// SIMATIC STEP 7 (V5.x) project parking2
// CPU: CPU 314C-2 DP
// station: Hardware
// station: SIMATIC 300(1)
// station: P_ADR_BUS
// program: S7 Program(2)

SYMBOL_TABLE
"res"	I 0.0	BOOL	// КжЮЭ ИСдЗге
"active"	I 0.5	BOOL	// ЭЪЗб УЗТ ИСдЗге
"enter"	I 0.6	BOOL	// ФУКн жСжПн
"exit"	I 0.7	BOOL	// ФУКн ОСжМн
"red light"	Q 0.0	BOOL
"yellow light"	Q 0.1	BOOL
"green light"	Q 0.2	BOOL
"light floor 1"	Q 1.0	BOOL
"light floor 2"	Q 1.1	BOOL
"light floor 3"	Q 1.2	BOOL
"parking is full"	Q 1.3	BOOL
"fan 1"	Q 1.4	BOOL	// floor 1
"fan 2"	Q 1.5	BOOL	// floor 1
"fan 3"	Q 1.6	BOOL	// floor 1
"fan 4"	Q 1.7	BOOL	// floor 1
"fan 5"	Q 2.0	BOOL	// floor 2
"fan 6"	Q 2.1	BOOL	// floor 2
"fan 7"	Q 2.2	BOOL	// floor 2
"fan 8"	Q 2.3	BOOL	// floor 2
"fan 9"	Q 2.4	BOOL	// floor 3
"fan 10"	Q 2.5	BOOL	// floor 3
"fan 11"	Q 2.6	BOOL	// floor 3
"fan 12"	Q 2.7	BOOL	// floor 3
END_SYMBOL_TABLE

ORGANIZATION_BLOCK OB 1
TITLE = "Main Program Sweep (Cycle)"
VERSION : 0.1
VAR_TEMP
  OB1_EV_CLASS : BYTE ;	//Bits 0-3 = 1 (Coming event), Bits 4-7 = 1 (Event class 1)
  OB1_SCAN_1 : BYTE ;	//1 (Cold restart scan 1 of OB 1), 3 (Scan 2-n of OB 1)
  OB1_PRIORITY : BYTE ;	//Priority of OB Execution
  OB1_OB_NUMBR : BYTE ;	//1 (Organization block 1, OB1)
  OB1_RESERVED_1 : BYTE ;	//Reserved for system
  OB1_RESERVED_2 : BYTE ;	//Reserved for system
  OB1_PREV_CYCLE : INT ;	//Cycle time of previous OB1 scan (milliseconds)
  OB1_MIN_CYCLE : INT ;	//Minimum cycle time of OB1 (milliseconds)
  OB1_MAX_CYCLE : INT ;	//Maximum cycle time of OB1 (milliseconds)
  OB1_DATE_TIME : DATE_AND_TIME ;	//Date and time OB1 started
END_VAR
BEGIN
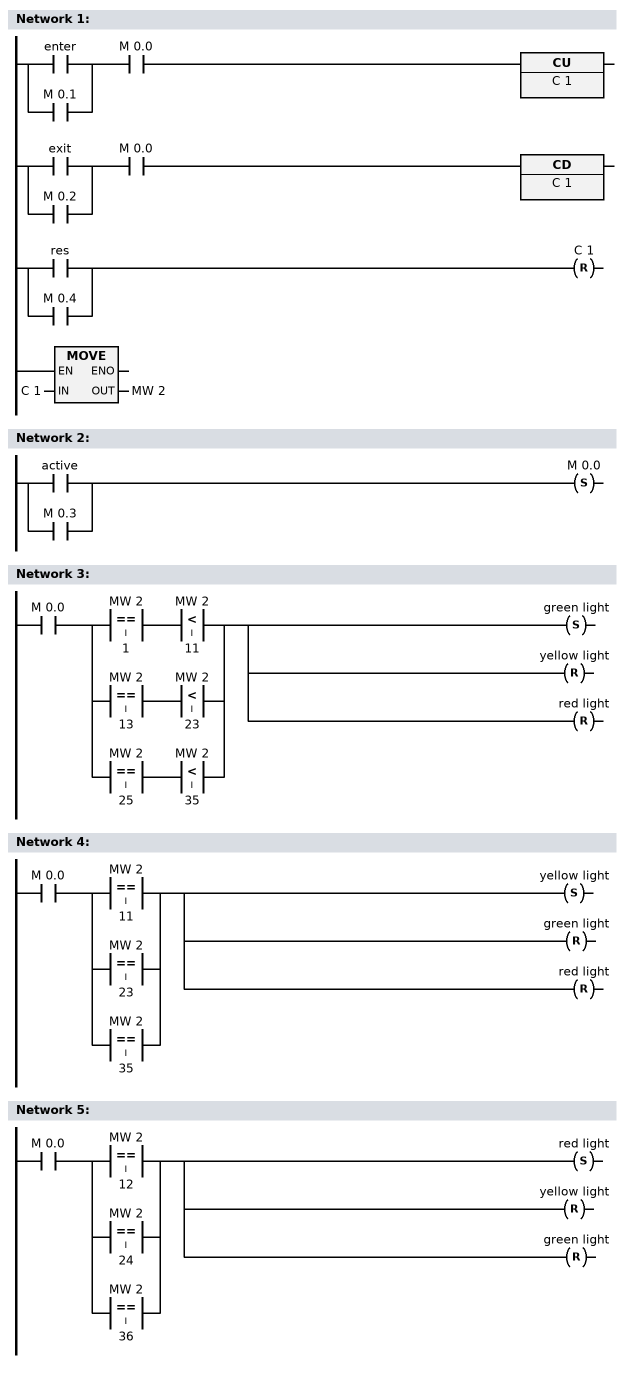
NETWORK
TITLE =
      A(;
      O     "enter";
      O     M 0.1;
      );
      A     M 0.0;
      CU    C 1;
      A(;
      O     "exit";
      O     M 0.2;
      );
      A     M 0.0;
      CD    C 1;
      NOP   0;
      NOP   0;
      A(;
      O     "res";
      O     M 0.4;
      );
      R     C 1;
      L     C 1;
      T     MW 2;
      NOP   0;
      NOP   0;
NETWORK
TITLE =
      O     "active";
      O     M 0.3;
      S     M 0.0;
NETWORK
TITLE =
      A     M 0.0;
      A(;
      A(;
      L     MW 2;
      L     1;
      ==I;
      );
      A(;
      L     MW 2;
      L     11;
      <I;
      );
      O;
      A(;
      L     MW 2;
      L     13;
      ==I;
      );
      A(;
      L     MW 2;
      L     23;
      <I;
      );
      O;
      A(;
      L     MW 2;
      L     25;
      ==I;
      );
      A(;
      L     MW 2;
      L     35;
      <I;
      );
      );
      S     "green light";
      R     "yellow light";
      R     "red light";
NETWORK
TITLE =
      A     M 0.0;
      A(;
      O(;
      L     MW 2;
      L     11;
      ==I;
      );
      O(;
      L     MW 2;
      L     23;
      ==I;
      );
      O(;
      L     MW 2;
      L     35;
      ==I;
      );
      );
      S     "yellow light";
      R     "green light";
      R     "red light";
NETWORK
TITLE =
      A     M 0.0;
      A(;
      O(;
      L     MW 2;
      L     12;
      ==I;
      );
      O(;
      L     MW 2;
      L     24;
      ==I;
      );
      O(;
      L     MW 2;
      L     36;
      ==I;
      );
      );
      S     "red light";
      R     "yellow light";
      R     "green light";
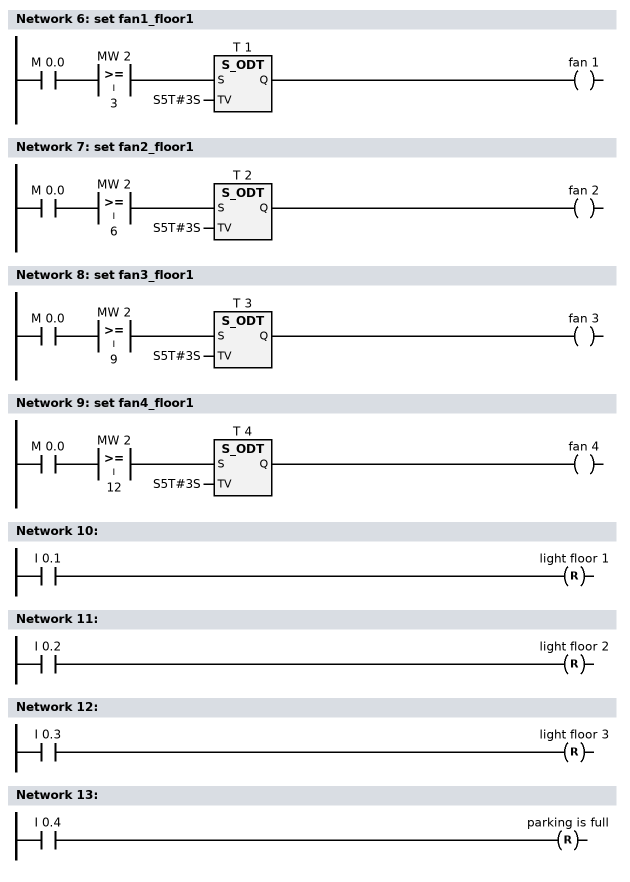
NETWORK
TITLE = set fan1_floor1
      A     M 0.0;
      A(;
      L     MW 2;
      L     3;
      >=I;
      );
      L     S5T#3S;
      SD    T 1;
      NOP   0;
      NOP   0;
      NOP   0;
      A     T 1;
      =     "fan 1";
NETWORK
TITLE = set fan2_floor1
      A     M 0.0;
      A(;
      L     MW 2;
      L     6;
      >=I;
      );
      L     S5T#3S;
      SD    T 2;
      NOP   0;
      NOP   0;
      NOP   0;
      A     T 2;
      =     "fan 2";
NETWORK
TITLE = set fan3_floor1
      A     M 0.0;
      A(;
      L     MW 2;
      L     9;
      >=I;
      );
      L     S5T#3S;
      SD    T 3;
      NOP   0;
      NOP   0;
      NOP   0;
      A     T 3;
      =     "fan 3";
NETWORK
TITLE = set fan4_floor1
      A     M 0.0;
      A(;
      L     MW 2;
      L     12;
      >=I;
      );
      L     S5T#3S;
      SD    T 4;
      NOP   0;
      NOP   0;
      NOP   0;
      A     T 4;
      =     "fan 4";
NETWORK
TITLE =
      A     I 0.1;
      R     "light floor 1";
NETWORK
TITLE =
      A     I 0.2;
      R     "light floor 2";
NETWORK
TITLE =
      A     I 0.3;
      R     "light floor 3";
NETWORK
TITLE =
      A     I 0.4;
      R     "parking is full";
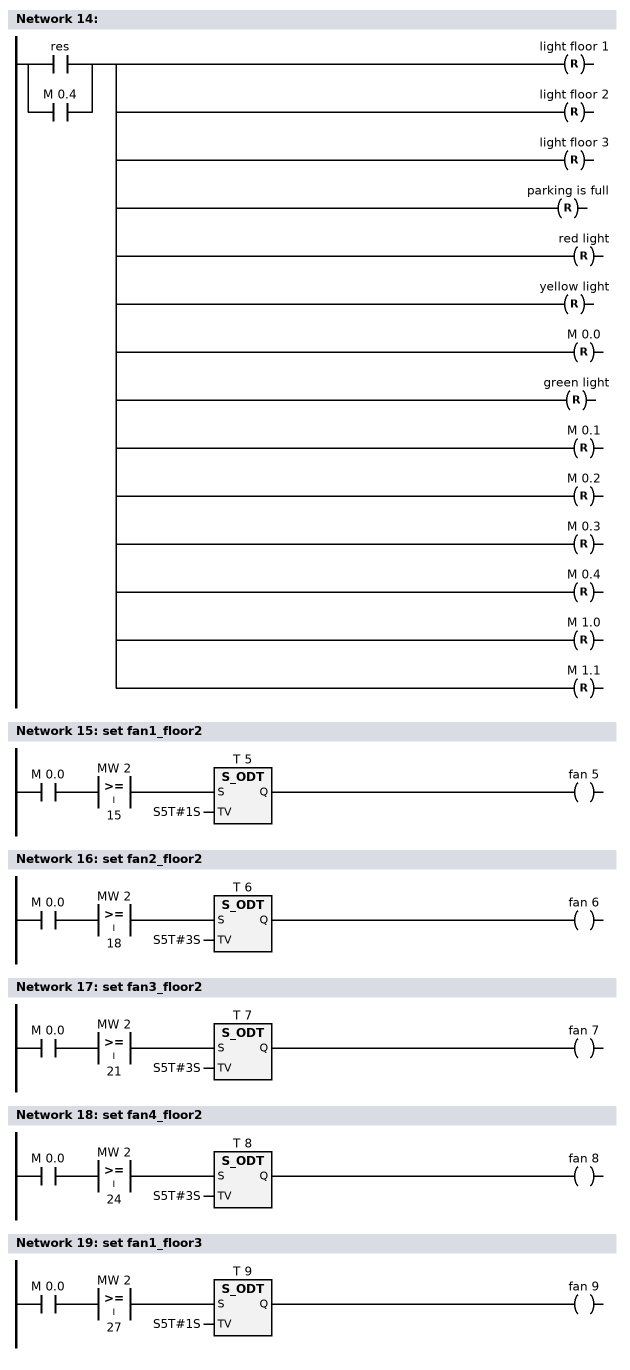
NETWORK
TITLE =
      O     "res";
      O     M 0.4;
      R     "light floor 1";
      R     "light floor 2";
      R     "light floor 3";
      R     "parking is full";
      R     "red light";
      R     "yellow light";
      R     M 0.0;
      R     "green light";
      R     M 0.1;
      R     M 0.2;
      R     M 0.3;
      R     M 0.4;
      R     M 1.0;
      R     M 1.1;
NETWORK
TITLE = set fan1_floor2
      A     M 0.0;
      A(;
      L     MW 2;
      L     15;
      >=I;
      );
      L     S5T#1S;
      SD    T 5;
      NOP   0;
      NOP   0;
      NOP   0;
      A     T 5;
      =     "fan 5";
NETWORK
TITLE = set fan2_floor2
      A     M 0.0;
      A(;
      L     MW 2;
      L     18;
      >=I;
      );
      L     S5T#3S;
      SD    T 6;
      NOP   0;
      NOP   0;
      NOP   0;
      A     T 6;
      =     "fan 6";
NETWORK
TITLE = set fan3_floor2
      A     M 0.0;
      A(;
      L     MW 2;
      L     21;
      >=I;
      );
      L     S5T#3S;
      SD    T 7;
      NOP   0;
      NOP   0;
      NOP   0;
      A     T 7;
      =     "fan 7";
NETWORK
TITLE = set fan4_floor2
      A     M 0.0;
      A(;
      L     MW 2;
      L     24;
      >=I;
      );
      L     S5T#3S;
      SD    T 8;
      NOP   0;
      NOP   0;
      NOP   0;
      A     T 8;
      =     "fan 8";
NETWORK
TITLE = set fan1_floor3
      A     M 0.0;
      A(;
      L     MW 2;
      L     27;
      >=I;
      );
      L     S5T#1S;
      SD    T 9;
      NOP   0;
      NOP   0;
      NOP   0;
      A     T 9;
      =     "fan 9";
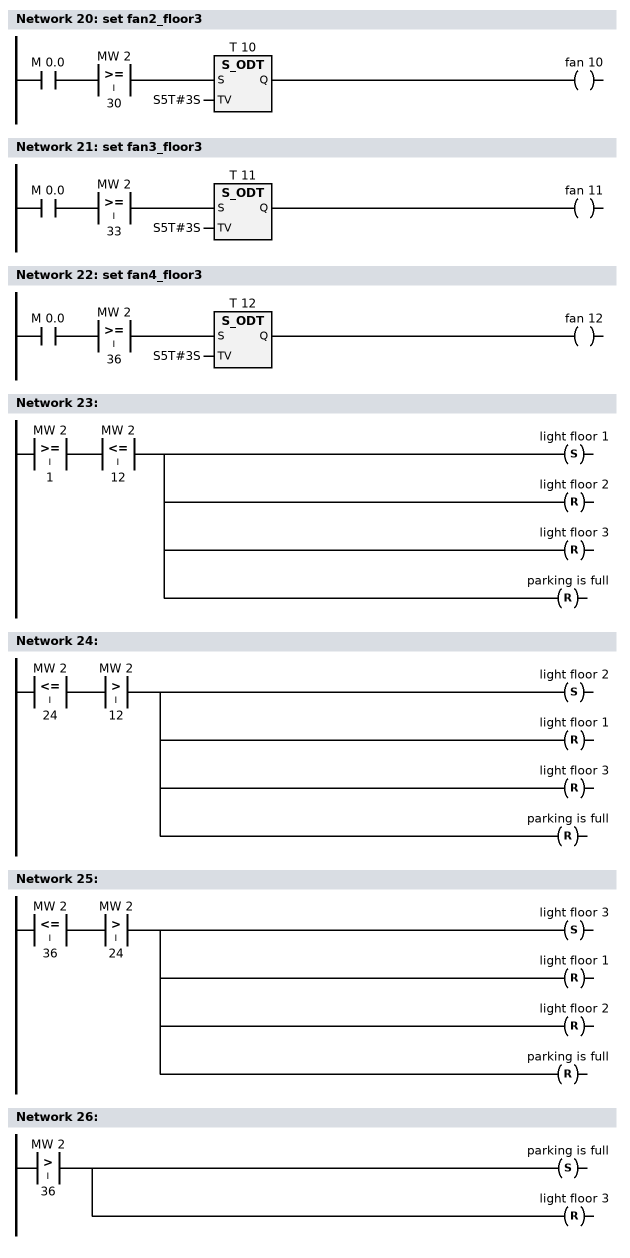
NETWORK
TITLE = set fan2_floor3
      A     M 0.0;
      A(;
      L     MW 2;
      L     30;
      >=I;
      );
      L     S5T#3S;
      SD    T 10;
      NOP   0;
      NOP   0;
      NOP   0;
      A     T 10;
      =     "fan 10";
NETWORK
TITLE = set fan3_floor3
      A     M 0.0;
      A(;
      L     MW 2;
      L     33;
      >=I;
      );
      L     S5T#3S;
      SD    T 11;
      NOP   0;
      NOP   0;
      NOP   0;
      A     T 11;
      =     "fan 11";
NETWORK
TITLE = set fan4_floor3
      A     M 0.0;
      A(;
      L     MW 2;
      L     36;
      >=I;
      );
      L     S5T#3S;
      SD    T 12;
      NOP   0;
      NOP   0;
      NOP   0;
      A     T 12;
      =     "fan 12";
NETWORK
TITLE =
      A(;
      L     MW 2;
      L     1;
      >=I;
      );
      A(;
      L     MW 2;
      L     12;
      <=I;
      );
      S     "light floor 1";
      R     "light floor 2";
      R     "light floor 3";
      R     "parking is full";
NETWORK
TITLE =
      A(;
      L     MW 2;
      L     24;
      <=I;
      );
      A(;
      L     MW 2;
      L     12;
      >I;
      );
      S     "light floor 2";
      R     "light floor 1";
      R     "light floor 3";
      R     "parking is full";
NETWORK
TITLE =
      A(;
      L     MW 2;
      L     36;
      <=I;
      );
      A(;
      L     MW 2;
      L     24;
      >I;
      );
      S     "light floor 3";
      R     "light floor 1";
      R     "light floor 2";
      R     "parking is full";
NETWORK
TITLE =
      L     MW 2;
      L     36;
      >I;
      S     "parking is full";
      R     "light floor 3";
END_ORGANIZATION_BLOCK
